{attribute addProperty BoxType "EK1122-0000-0018"}
{attribute addProperty Id "Beckhoff_EPP4xxxsub_EK1100EK1100_179A0949162A_0001_EPP4174_0002_0016EPP4174_253CF8AE15219A_0002_EPP4174_0002_0017EPP4174_253CF8AE15219A_0003_EPP4314_1002_0016EPP4314_43F10CD122428A_0004_EPP4374_0002_0016EPP4374_D464211E19224A_0005_EPP4374_0002_0017EPP4374_D464211E19224A_0006_EPP4374_0002_0018EPP4374_D464211E19224A_0007_EPP4374_0002_0019EPP4374_D464211E19224"}
{attribute addProperty CRC "1006956348"}
{attribute addProperty SizeInBites "1312"}
{attribute addProperty SizeInBytes "164"}
TYPE Beckhoff_EPP4xxxEK1122_3C04EF3C EXTENDS EK1122_179A0949 :
STRUCT
	{attribute addProperty Name "Beckhoff_EPP4xxxsub_EK1100"}
	Beckhoff_EPP4xxxsub_EK1100 : EK1100_179A0949;
	{attribute addProperty Name "A_0001_EPP4174_0002_0016"}
	A_0001_EPP4174_0002_0016 : EPP4174_253CF8AE;
	{attribute addProperty Name "A_0002_EPP4174_0002_0017"}
	A_0002_EPP4174_0002_0017 : EPP4174_253CF8AE;
	{attribute addProperty Name "A_0003_EPP4314_1002_0016"}
	A_0003_EPP4314_1002_0016 : EPP4314_43F10CD1;
	{attribute addProperty Name "A_0004_EPP4374_0002_0016"}
	A_0004_EPP4374_0002_0016 : EPP4374_D464211E;
	{attribute addProperty Name "A_0005_EPP4374_0002_0017"}
	A_0005_EPP4374_0002_0017 : EPP4374_D464211E;
	{attribute addProperty Name "A_0006_EPP4374_0002_0018"}
	A_0006_EPP4374_0002_0018 : EPP4374_D464211E;
	{attribute addProperty Name "A_0007_EPP4374_0002_0019"}
	A_0007_EPP4374_0002_0019 : EPP4374_D464211E;
END_STRUCT
END_TYPE

(* stored: Version 1.2.0.0, ProductVersion 3.1.4024.9
   DUT Beckhoff_EPP4xxxEK1122_3C04EF3C: Id {360a85fd-27fb-43fb-a6a1-997a5dd32a55} *)
